TYPE ST_ComponentBase_Config :
    STRUCT
        Name : STRING;
    END_STRUCT
END_TYPE

(* stored: Version 1.1.0.1, ProductVersion 3.1.4024.12
   DUT ST_ComponentBase_Config: Id {3f71f39c-219c-40af-b645-bb22eb1c678f} *)
